(* IEC 61131-3 sources: programs/VI-54/VI-54_20171205/VI-54_20171205/Stations/Screen/LseClass170718/Class/Position, 1 file *)

(* ---- Position.st ---- *)
(*!
<Class
	Name               = "Position"
	Revision           = "0.0"
	RealtimeTask       = "false"
	CyclicTask         = "false"
	BackgroundTask     = "false"
	Sigmatek           = "false"
	OSInterface        = "false"
	HighPriority       = "false"
	Automatic          = "false"
	UpdateMode         = "Prescan"
	SharedCommandTable = "true"
	Objectsize         = "(540,120)">
	<Channels>
		<Server Name="Nbr" Visualized="true" Initialize="false" WriteProtected="true" Retentive="false"/>
		<Server Name="Rpos" Visualized="true" Initialize="false" WriteProtected="false" Retentive="false"/>
		<Server Name="Xpos" Visualized="true" Initialize="false" WriteProtected="false" Retentive="false"/>
		<Server Name="Ypos" Visualized="true" Initialize="false" WriteProtected="false" Retentive="false"/>
		<Server Name="Zpos" Visualized="true" Initialize="false" WriteProtected="false" Retentive="false"/>
		<Client Name="Next" Required="false" Internal="false"/>
	</Channels>
</Class>
*)
Position : CLASS
  //Servers:
	Nbr 	: SvrChCmd_DINT;
	Xpos 	: SvrCh_DINT;
	Zpos 	: SvrCh_DINT;
	Rpos 	: SvrCh_DINT;
	Ypos 	: SvrCh_DINT;
  //Clients:
	Next 	: CltChCmd_Position;
  //Variables:
		ReceptPtr 	: ^RecipeStr;
  //Functions:

	FUNCTION GLOBAL PosNbr
		VAR_INPUT
			inpNbr 	: DINT;
		END_VAR;

	FUNCTION GLOBAL PosData
		VAR_INPUT
			inpData 	: RobotPosStr;
			inpNbr 	: DINT;
		END_VAR;

	FUNCTION GLOBAL SetRecipePtr
		VAR_INPUT
			Ptr 	: ^RecipeStr;
		END_VAR;

	FUNCTION VIRTUAL GLOBAL Xpos::Write
		VAR_INPUT
			input (EAX) 	: DINT;
		END_VAR
		VAR_OUTPUT
			result (EAX) 	: DINT;
		END_VAR;

	FUNCTION VIRTUAL GLOBAL Zpos::Write
		VAR_INPUT
			input (EAX) 	: DINT;
		END_VAR
		VAR_OUTPUT
			result (EAX) 	: DINT;
		END_VAR;

	FUNCTION VIRTUAL GLOBAL Rpos::Write
		VAR_INPUT
			input (EAX) 	: DINT;
		END_VAR
		VAR_OUTPUT
			result (EAX) 	: DINT;
		END_VAR;

	FUNCTION VIRTUAL GLOBAL Ypos::Write
		VAR_INPUT
			input (EAX) 	: DINT;
		END_VAR
		VAR_OUTPUT
			result (EAX) 	: DINT;
		END_VAR;
  //Tables:
	FUNCTION @STD
		VAR_OUTPUT
			ret_code	: CONFSTATES;
		END_VAR;
	FUNCTION GLOBAL TAB @CT_;
END_CLASS;

FUNCTION GLOBAL Position::PosNbr
	VAR_INPUT
		inpNbr 	: DINT;
	END_VAR

  Nbr := inpNbr;

  if IsClientConnected(#Next) then
    Next.PosNbr(inpNbr:= inpNbr + 1);
  end_if;

END_FUNCTION

FUNCTION GLOBAL Position::SetRecipePtr
	VAR_INPUT
		Ptr 	: ^RecipeStr;
	END_VAR

  ReceptPtr := Ptr;
  if IsClientConnected(#Next) then
    Next.SetRecipePtr(Ptr:= ReceptPtr);
  end_if;

END_FUNCTION

FUNCTION GLOBAL Position::PosData
	VAR_INPUT
		inpData 	: RobotPosStr;
		inpNbr 	: DINT;
	END_VAR

  if inpNbr = Nbr then
    Xpos    := inpData.Xpos;
    Ypos    := inpData.Ypos;
    Zpos    := inpData.Zpos;
    Rpos    := inpData.Rpos;
  elsif IsClientConnected(#Next) then
    Next.PosData(inpData:= inpData, inpNbr:= inpNbr);
  end_if;

END_FUNCTION

FUNCTION VIRTUAL GLOBAL Position::Xpos::Write
	VAR_INPUT
		input (EAX) 	: DINT;
	END_VAR
	VAR_OUTPUT
		result (EAX) 	: DINT;
	END_VAR

	Xpos := input;
  ReceptPtr^.RobotPositions[Nbr].Xpos := Xpos;
	result := Xpos;

END_FUNCTION

FUNCTION VIRTUAL GLOBAL Position::Zpos::Write
	VAR_INPUT
		input (EAX) 	: DINT;
	END_VAR
	VAR_OUTPUT
		result (EAX) 	: DINT;
	END_VAR

	Zpos := input;
  ReceptPtr^.RobotPositions[Nbr].Zpos := Zpos;
	result := Zpos;

END_FUNCTION

FUNCTION VIRTUAL GLOBAL Position::Rpos::Write
	VAR_INPUT
		input (EAX) 	: DINT;
	END_VAR
	VAR_OUTPUT
		result (EAX) 	: DINT;
	END_VAR

	Rpos := input;
  ReceptPtr^.RobotPositions[Nbr].Rpos := Rpos;
	result := Rpos;

END_FUNCTION

FUNCTION VIRTUAL GLOBAL Position::Ypos::Write
	VAR_INPUT
		input (EAX) 	: DINT;
	END_VAR
	VAR_OUTPUT
		result (EAX) 	: DINT;
	END_VAR

	Ypos := input;
  ReceptPtr^.RobotPositions[Nbr].Ypos := Ypos;
	result := Ypos;

END_FUNCTION
